FUNCTION AmsNetID_TO_TAmsNetID : T_AmsNetID
VAR_INPUT
	sNetId 						:	AmsNetID;
END_VAR
VAR
END_VAR

AmsNetID_TO_TAmsNetID := CONCAT(BYTE_TO_STRING(sNetId[0]),'.');
AmsNetID_TO_TAmsNetID := CONCAT(AmsNetID_TO_TAmsNetID, BYTE_TO_STRING(sNetId[1]));	
AmsNetID_TO_TAmsNetID := CONCAT(AmsNetID_TO_TAmsNetID,'.');
AmsNetID_TO_TAmsNetID := CONCAT(AmsNetID_TO_TAmsNetID, BYTE_TO_STRING(sNetId[2]));	
AmsNetID_TO_TAmsNetID := CONCAT(AmsNetID_TO_TAmsNetID,'.');
AmsNetID_TO_TAmsNetID := CONCAT(AmsNetID_TO_TAmsNetID, BYTE_TO_STRING(sNetId[3]));	
AmsNetID_TO_TAmsNetID := CONCAT(AmsNetID_TO_TAmsNetID,'.');
AmsNetID_TO_TAmsNetID := CONCAT(AmsNetID_TO_TAmsNetID, BYTE_TO_STRING(sNetId[4]));	
AmsNetID_TO_TAmsNetID := CONCAT(AmsNetID_TO_TAmsNetID,'.');
AmsNetID_TO_TAmsNetID := CONCAT(AmsNetID_TO_TAmsNetID, BYTE_TO_STRING(sNetId[5]));

END_FUNCTION

(* stored: Version 1.1.0.1, ProductVersion 3.1.4020.12
   POU AmsNetID_TO_TAmsNetID: Id {5801596a-d2ca-4f92-b341-d7bee2be61c2}, SpecialFunc None *)
